FUNCTION_BLOCK FB_CRYO_TEMPERATURES
VAR_INPUT
END_VAR
VAR_OUTPUT
END_VAR
VAR
END_VAR

END_FUNCTION_BLOCK

(* stored: Version 1.1.0.1, ProductVersion 3.1.4024.12
   POU FB_CRYO_TEMPERATURES: Id {da3db0a8-7555-40f7-8a65-0f78d8431970}, SpecialFunc None *)
